ABB RobotStudio station: IRB1600_20220616-161156.rsstn

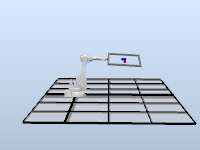
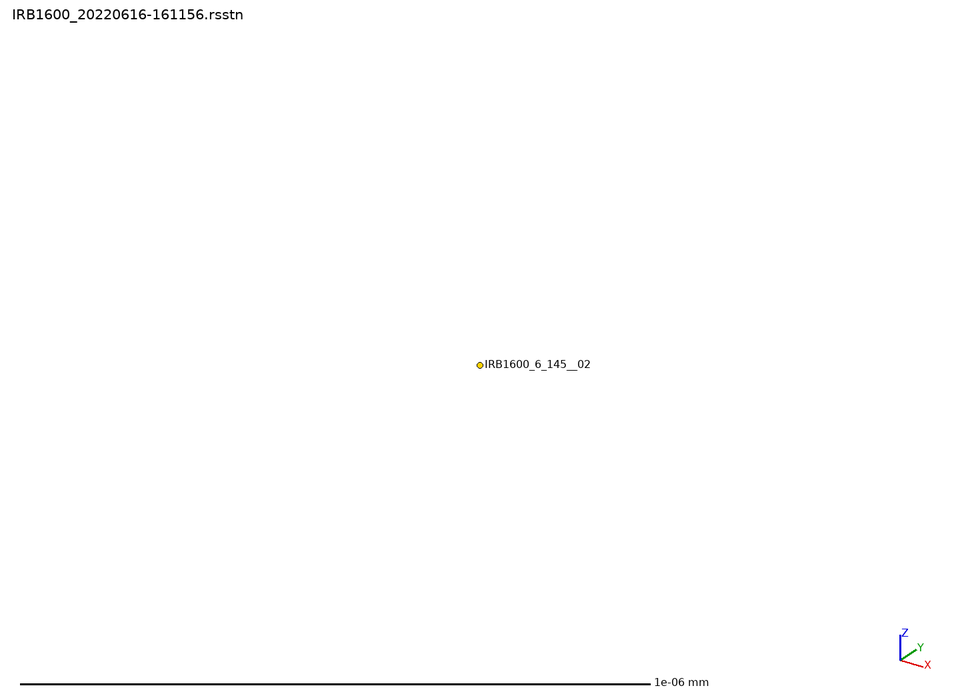
[picture v1: parts stored in the station drawn from their meshes, with robot base, taught points and paths (robot models come from the ABB library and are not in the file)]
Station Solution1 (saved by RobotStudio 22.1.9826.0)
Controller IRB1600_6_145
  mechanical unit ROB_1: IRB1600_6_145__02, 6 joints, base frame (0, 0, 0) mm
Layout (positions relative to the parent item):
  - IRB1600_6_145__02 [mechanism, from Robots\IRB1600_6_145_G_02.rslib] at (0, 0, 0) mm; joint values [0.005, 0.184, -0.1478, -3.3944, -0.021, 3.6208] (rad or m)
  - flange_connector [part, from Tools\IsoPlate_small_Binzel.rslib] at (942.53, 4.38, 1149.32) mm, rotated rx 104.17 ry 76.65 rz 103.78 deg
  - plane [part] at (1451.34, 5.61, 1125.62) mm, rotated rx 167.04 ry -3.24 rz 179.98 deg, size 1000 x 1000 x 50 mm
  - Frame_1 [frame]
  - Frame_2 [frame] at (-23.65, -1.83, 250.36) mm
Attachment: flange_connector is attached to IRB1600_6_145__02 / Link6
Attachment: plane is attached to flange_connector
Targets, tools, work objects and paths stored in the station, written as RAPID:
! task T_ROB1
MODULE Module1
  LOCAL PERS wobjdata egm_wobj:=[FALSE,TRUE,"",[[0,0,0],[1,0,0,0]],[[0,0,0],[1,0,0,0]]];
  PROC main()
    ConfJ \On;
  ENDPROC
  PROC EGM_CARTESIAN_MOVE()
    WaitTime 2;
  ENDPROC
  PROC RAPID_MOVE()
  ENDPROC
ENDMODULE

! task T_ROB1
MODULE CalibData
  TASK PERS tooldata Tooldata_4:=[TRUE,[[0,0,0],[1,0,0,0]],[1,[0,0,1],[1,0,0,0],0,0,0]];
  TASK PERS tooldata Tooldata_5:=[TRUE,[[0,0,0],[1,0,0,0]],[1,[0,0,1],[1,0,0,0],0,0,0]];
  TASK PERS tooldata Tooldata_6:=[TRUE,[[0,0,0],[1,0,0,0]],[1,[0,0,1],[1,0,0,0],0,0,0]];
  TASK PERS tooldata Tooldata_7:=[TRUE,[[-23.772999698,2.161000196,740.120999999],[0.707106781,0,-0.707106781,0]],[1,[0,0,1],[1,0,0,0],0,0,0]];
  TASK PERS wobjdata Workobject_2:=[FALSE,TRUE,"ROB_1",[[-55.133477186,-6.202200727,258.13059393],[1,0,0,0]],[[0,0,0],[1,0,0,0]]];
  TASK PERS tooldata Tooldata_9:=[TRUE,[[20.616002648,0.899999913,497.265999882],[0.707106781,-0.000000002,-0.707106781,0]],[1,[0,0,1],[1,0,0,0],0,0,0]];
ENDMODULE

